/// configuration data that is used during boot to configure the Units equipment
TYPE PickerDataConfig :
STRUCT
  Simulated : BOOL;
END_STRUCT
END_TYPE

(* stored: Version 1.1.0.1
   DUT PickerDataConfig: Id {7205ea24-b5d3-405b-8359-986e7345fef2} *)
